(* CODESYS project Cooking chamber.project

Project tree, tasks and I/O mapping:
  Device : L-force Panel Controller p300 Logic, Lenze, order no. LPC 1000, version 3.8.0.0
    application Application
      libraries: L_PLCDataManagerAccess, 3.0.0.0 (Lenze); L_PLCLoggingAccess, 3.3.0.0 (Lenze); L_Util, 3.3.0.0 (Lenze); CAA CiA 405, 3.5.3.0 (CAA Technical Workgroup)
      task MainTask (cyclic, interval t#10ms, priority 1) calls Main
      Programs/
        program Main [ST]
        Functions/
          function Timer_convert [ST]
          function block Chamber_controller [ST]
          function block Chamber_program [ST]
          function Humidity_convert [ST]
          function block Sound_controller [ST]
          function block Alarm_controller [ST]
        Routines/
          program Controller [ST]
        System/
          program Analog_controller [ST]
      Variables/
        global variables Global
        global variables Settings
        global variables Recipes
      Symbols/
        Symbols
    CANbus : CANbus, Lenze, version 2.0.0.0
      CANopen_Manager : CANopen_Manager, Lenze, version 3.12.0.0
          settings: Sync CycleTime in Microseconds = 10000; Enable Sync generation = TRUE; Heartbeat Node ID = 63; Can Open Node ID = 63; ConfigVersion = 50659584
        EPM_S110 : EPM-S110, Lenze, order no. EPM-S110, version 1.14.0.5
            settings: General Options.Reset Node = FALSE; NODEIDSAVED = 1; SDO Timeout = 1000000; EXPERTSETTINGS = TRUE; Sync-General Parameters.Communication Cycle Period = 16#00002710 usec; Synchronous Window Length = 16#000004B0; Emergency-General Parameters.Emergency enabled = FALSE; Settings.COBID = 16#00000201; Settings.Transmission Type = 16#FF; Settings.available PDO-Parameter.Inhibit Time available = FALSE; Settings.available PDO-Parameter.Event Timer available = FALSE; Settings.Inhibit Time = 0; Settings.Event Timer = 0; Generic COBID = '$NODEID+16#0200'; Settings.COBID = 16#00000181; Settings.Transmission Type = 16#01; Settings.available PDO-Parameter.Inhibit Time available = TRUE; Settings.available PDO-Parameter.Event Timer available = TRUE; Settings.Inhibit Time = 0; Settings.Event Timer = 0; Generic COBID = '$NODEID+16#0180'; Settings.COBID = 16#00000281; Settings.Transmission Type = 16#01; Settings.available PDO-Parameter.Inhibit Time available = TRUE; Settings.available PDO-Parameter.Event Timer available = TRUE; Settings.Inhibit Time = 0; Settings.Event Timer = 0; Generic COBID = '$NODEID+16#0280'; Settings.COBID = 16#00000381; Settings.Transmission Type = 16#01; Settings.available PDO-Parameter.Inhibit Time available = TRUE; Settings.available PDO-Parameter.Event Timer available = TRUE; Settings.Inhibit Time = 0; Settings.Event Timer = 0; Generic COBID = '$NODEID+16#0380'; Setting /state digital Output : EPM_S302_DO8_DC24V_5A_02.Index = 16#6200; Setting /state digital Output : EPM_S302_DO8_DC24V_5A_02.Subindex = 16#01; Setting /state digital Output : EPM_S302_DO8_DC24V_5A_02.ObjectLength = 8; Setting /state digital Output : EPM_S302_DO8_DC24V_5A_03.Index = 16#6200; Setting /state digital Output : EPM_S302_DO8_DC24V_5A_03.Subindex = 16#02;
              Setting /state digital Output : EPM_S302_DO8_DC24V_5A_03.ObjectLength = 8; State digital input : EPM_S202_DI8_DC24V_00.Index = 16#6000; State digital input : EPM_S202_DI8_DC24V_00.Subindex = 16#01; State digital input : EPM_S202_DI8_DC24V_00.ObjectLength = 8; State digital input : EPM_S202_DI8_DC24V_01.Index = 16#6000; State digital input : EPM_S202_DI8_DC24V_01.Subindex = 16#02; State digital input : EPM_S202_DI8_DC24V_01.ObjectLength = 8; Read analog Input : EPM_S404_AI4_16Bit_Resistor_04.Index = 16#6401; Read analog Input : EPM_S404_AI4_16Bit_Resistor_04.Subindex = 16#01; Read analog Input : EPM_S404_AI4_16Bit_Resistor_04.ObjectLength = 16; Read analog Input : EPM_S404_AI4_16Bit_Resistor_04.Index = 16#6401; Read analog Input : EPM_S404_AI4_16Bit_Resistor_04.Subindex = 16#02; Read analog Input : EPM_S404_AI4_16Bit_Resistor_04.ObjectLength = 16; Read analog Input : EPM_S404_AI4_16Bit_Resistor_04.Index = 16#6401; Read analog Input : EPM_S404_AI4_16Bit_Resistor_04.Subindex = 16#03; Read analog Input : EPM_S404_AI4_16Bit_Resistor_04.ObjectLength = 16; Read analog Input : EPM_S404_AI4_16Bit_Resistor_04.Index = 16#6401; Read analog Input : EPM_S404_AI4_16Bit_Resistor_04.Subindex = 16#04; Read analog Input : EPM_S404_AI4_16Bit_Resistor_04.ObjectLength = 16; Read analog Input : EPM_S404_AI4_16Bit_Resistor_05.Index = 16#6401; Read analog Input : EPM_S404_AI4_16Bit_Resistor_05.Subindex = 16#05; Read analog Input : EPM_S404_AI4_16Bit_Resistor_05.ObjectLength = 16; Read analog Input : EPM_S404_AI4_16Bit_Resistor_05.Index = 16#6401; Read analog Input : EPM_S404_AI4_16Bit_Resistor_05.Subindex = 16#06; Read analog Input : EPM_S404_AI4_16Bit_Resistor_05.ObjectLength = 16; Read analog Input : EPM_S404_AI4_16Bit_Resistor_05.Index = 16#6401; Read analog Input : EPM_S404_AI4_16Bit_Resistor_05.Subindex = 16#07; Read analog Input : EPM_S404_AI4_16Bit_Resistor_05.ObjectLength = 16; Read analog Input : EPM_S404_AI4_16Bit_Resistor_05.Index = 16#6401; Read analog Input : EPM_S404_AI4_16Bit_Resistor_05.Subindex = 16#08; Read analog Input : EPM_S404_AI4_16Bit_Resistor_05.ObjectLength = 16; SDO List.Set COB-ID sync.Index = 16#1005; SDO List.Set COB-ID sync.Subindex = 16#00; SDO List.Set COB-ID sync.Value = 16#80000080; SDO List.Set COB-ID sync.Size = 32; SDO List.Set COB-ID sync.AbortIfError = FALSE; SDO List.Set COB-ID sync.JumpToLine = FALSE; SDO List.Set COB-ID sync.Line = 0; SDO List.Set synchronous window length.Index = 16#1007; SDO List.Set synchronous window length.Subindex = 16#00;
              SDO List.Set synchronous window length.Value = 16#000004B0; SDO List.Set synchronous window length.Size = 32; SDO List.Set synchronous window length.AbortIfError = FALSE; SDO List.Set synchronous window length.JumpToLine = FALSE; SDO List.Set synchronous window length.Line = 0; SDO List.Set Guardtime.Index = 16#100C; SDO List.Set Guardtime.Subindex = 16#00; SDO List.Set Guardtime.Value = 16#00000000; SDO List.Set Guardtime.Size = 16; SDO List.Set Guardtime.AbortIfError = FALSE; SDO List.Set Guardtime.JumpToLine = FALSE; SDO List.Set Guardtime.Line = 0; SDO List.Set Lifetime.Index = 16#100D; SDO List.Set Lifetime.Subindex = 16#00; SDO List.Set Lifetime.Value = 16#00000000; SDO List.Set Lifetime.Size = 8; SDO List.Set Lifetime.AbortIfError = FALSE; SDO List.Set Lifetime.JumpToLine = FALSE; SDO List.Set Lifetime.Line = 0; SDO List.Set Heartbeat Consumer.Index = 16#1016; SDO List.Set Heartbeat Consumer.Subindex = 16#01; SDO List.Set Heartbeat Consumer.Value = 0; SDO List.Set Heartbeat Consumer.Size = 32; SDO List.Set Heartbeat Consumer.AbortIfError = FALSE; SDO List.Set Heartbeat Consumer.JumpToLine = FALSE; SDO List.Set Heartbeat Consumer.Line = 0; SDO List.Set Heartbeat Consumer.Index = 16#1016; SDO List.Set Heartbeat Consumer.Subindex = 16#02; SDO List.Set Heartbeat Consumer.Value = 0; SDO List.Set Heartbeat Consumer.Size = 32; SDO List.Set Heartbeat Consumer.AbortIfError = FALSE; SDO List.Set Heartbeat Consumer.JumpToLine = FALSE; SDO List.Set Heartbeat Consumer.Line = 0; SDO List.Set Heartbeat Consumer.Index = 16#1016; SDO List.Set Heartbeat Consumer.Subindex = 16#03; SDO List.Set Heartbeat Consumer.Value = 0; SDO List.Set Heartbeat Consumer.Size = 32; SDO List.Set Heartbeat Consumer.AbortIfError = FALSE; SDO List.Set Heartbeat Consumer.JumpToLine = FALSE; SDO List.Set Heartbeat Consumer.Line = 0;
              SDO List.Set Heartbeat Consumer.Index = 16#1016; SDO List.Set Heartbeat Consumer.Subindex = 16#04; SDO List.Set Heartbeat Consumer.Value = 0; SDO List.Set Heartbeat Consumer.Size = 32; SDO List.Set Heartbeat Consumer.AbortIfError = FALSE; SDO List.Set Heartbeat Consumer.JumpToLine = FALSE; SDO List.Set Heartbeat Consumer.Line = 0; SDO List.Set Heartbeat Consumer.Index = 16#1016; SDO List.Set Heartbeat Consumer.Subindex = 16#05; SDO List.Set Heartbeat Consumer.Value = 0; SDO List.Set Heartbeat Consumer.Size = 32; SDO List.Set Heartbeat Consumer.AbortIfError = FALSE; SDO List.Set Heartbeat Consumer.JumpToLine = FALSE; SDO List.Set Heartbeat Consumer.Line = 0; SDO List.Set Heartbeat Producer.Index = 16#1017; SDO List.Set Heartbeat Producer.Subindex = 16#00; SDO List.Set Heartbeat Producer.Value = 16#00000000; SDO List.Set Heartbeat Producer.Size = 16; SDO List.Set Heartbeat Producer.AbortIfError = FALSE; SDO List.Set Heartbeat Producer.JumpToLine = FALSE; SDO List.Set Heartbeat Producer.Line = 0; SDO List.Disable PDO.Index = 16#1400; SDO List.Disable PDO.Subindex = 16#01; SDO List.Disable PDO.Value = 16#80000201; SDO List.Disable PDO.Size = 32; SDO List.Disable PDO.AbortIfError = FALSE; SDO List.Disable PDO.JumpToLine = FALSE; SDO List.Disable PDO.Line = 0; SDO List.Set transmission type.Index = 16#1400; SDO List.Set transmission type.Subindex = 16#02; SDO List.Set transmission type.Value = 16#FF; SDO List.Set transmission type.Size = 8; SDO List.Set transmission type.AbortIfError = FALSE; SDO List.Set transmission type.JumpToLine = FALSE; SDO List.Set transmission type.Line = 0; SDO List.Clear pdo mapping.Index = 16#1600; SDO List.Clear pdo mapping.Subindex = 16#00; SDO List.Clear pdo mapping.Value = 16#0; SDO List.Clear pdo mapping.Size = 8; SDO List.Clear pdo mapping.AbortIfError = FALSE;
              SDO List.Clear pdo mapping.JumpToLine = FALSE; SDO List.Clear pdo mapping.Line = 0; SDO List.Set Mapping.Index = 16#1600; SDO List.Set Mapping.Subindex = 16#01; SDO List.Set Mapping.Value = 16#62000108; SDO List.Set Mapping.Size = 32; SDO List.Set Mapping.AbortIfError = FALSE; SDO List.Set Mapping.JumpToLine = FALSE; SDO List.Set Mapping.Line = 0; SDO List.Set Mapping.Index = 16#1600; SDO List.Set Mapping.Subindex = 16#02; SDO List.Set Mapping.Value = 16#62000208; SDO List.Set Mapping.Size = 32; SDO List.Set Mapping.AbortIfError = FALSE; SDO List.Set Mapping.JumpToLine = FALSE; SDO List.Set Mapping.Line = 0; SDO List.Set number of mappings.Index = 16#1600; SDO List.Set number of mappings.Subindex = 16#00; SDO List.Set number of mappings.Value = 16#02; SDO List.Set number of mappings.Size = 8; SDO List.Set number of mappings.AbortIfError = FALSE; SDO List.Set number of mappings.JumpToLine = FALSE; SDO List.Set number of mappings.Line = 0; SDO List.Set and enable COB-ID.Index = 16#1400; SDO List.Set and enable COB-ID.Subindex = 16#01; SDO List.Set and enable COB-ID.Value = 16#00000201; SDO List.Set and enable COB-ID.Size = 32; SDO List.Set and enable COB-ID.AbortIfError = FALSE; SDO List.Set and enable COB-ID.JumpToLine = FALSE; SDO List.Set and enable COB-ID.Line = 0; SDO List.Disable PDO.Index = 16#1800; SDO List.Disable PDO.Subindex = 16#01; SDO List.Disable PDO.Value = 16#80000181; SDO List.Disable PDO.Size = 32; SDO List.Disable PDO.AbortIfError = FALSE; SDO List.Disable PDO.JumpToLine = FALSE; SDO List.Disable PDO.Line = 0; SDO List.Set transmission type.Index = 16#1800; SDO List.Set transmission type.Subindex = 16#02; SDO List.Set transmission type.Value = 16#01;
              SDO List.Set transmission type.Size = 8; SDO List.Set transmission type.AbortIfError = FALSE; SDO List.Set transmission type.JumpToLine = FALSE; SDO List.Set transmission type.Line = 0; SDO List.Set inhibit time.Index = 16#1800; SDO List.Set inhibit time.Subindex = 16#03; SDO List.Set inhibit time.Value = 16#0000; SDO List.Set inhibit time.Size = 16; SDO List.Set inhibit time.AbortIfError = FALSE; SDO List.Set inhibit time.JumpToLine = FALSE; SDO List.Set inhibit time.Line = 0; SDO List.Set event time.Index = 16#1800; SDO List.Set event time.Subindex = 16#05; SDO List.Set event time.Value = 16#0000; SDO List.Set event time.Size = 16; SDO List.Set event time.AbortIfError = FALSE; SDO List.Set event time.JumpToLine = FALSE; SDO List.Set event time.Line = 0; SDO List.Clear pdo mapping.Index = 16#1A00; SDO List.Clear pdo mapping.Subindex = 16#00; SDO List.Clear pdo mapping.Value = 16#0; SDO List.Clear pdo mapping.Size = 8; SDO List.Clear pdo mapping.AbortIfError = FALSE; SDO List.Clear pdo mapping.JumpToLine = FALSE; SDO List.Clear pdo mapping.Line = 0; SDO List.Set Mapping.Index = 16#1A00; SDO List.Set Mapping.Subindex = 16#01; SDO List.Set Mapping.Value = 16#60000108; SDO List.Set Mapping.Size = 32; SDO List.Set Mapping.AbortIfError = FALSE; SDO List.Set Mapping.JumpToLine = FALSE; SDO List.Set Mapping.Line = 0; SDO List.Set Mapping.Index = 16#1A00; SDO List.Set Mapping.Subindex = 16#02; SDO List.Set Mapping.Value = 16#60000208; SDO List.Set Mapping.Size = 32; SDO List.Set Mapping.AbortIfError = FALSE; SDO List.Set Mapping.JumpToLine = FALSE; SDO List.Set Mapping.Line = 0; SDO List.Set number of mappings.Index = 16#1A00;
              SDO List.Set number of mappings.Subindex = 16#00; SDO List.Set number of mappings.Value = 16#02; SDO List.Set number of mappings.Size = 8; SDO List.Set number of mappings.AbortIfError = FALSE; SDO List.Set number of mappings.JumpToLine = FALSE; SDO List.Set number of mappings.Line = 0; SDO List.Set and enable COB-ID.Index = 16#1800; SDO List.Set and enable COB-ID.Subindex = 16#01; SDO List.Set and enable COB-ID.Value = 16#00000181; SDO List.Set and enable COB-ID.Size = 32; SDO List.Set and enable COB-ID.AbortIfError = FALSE; SDO List.Set and enable COB-ID.JumpToLine = FALSE; SDO List.Set and enable COB-ID.Line = 0; SDO List.Disable PDO.Index = 16#1801; SDO List.Disable PDO.Subindex = 16#01; SDO List.Disable PDO.Value = 16#80000281; SDO List.Disable PDO.Size = 32; SDO List.Disable PDO.AbortIfError = FALSE; SDO List.Disable PDO.JumpToLine = FALSE; SDO List.Disable PDO.Line = 0; SDO List.Set transmission type.Index = 16#1801; SDO List.Set transmission type.Subindex = 16#02; SDO List.Set transmission type.Value = 16#01; SDO List.Set transmission type.Size = 8; SDO List.Set transmission type.AbortIfError = FALSE; SDO List.Set transmission type.JumpToLine = FALSE; SDO List.Set transmission type.Line = 0; SDO List.Set inhibit time.Index = 16#1801; SDO List.Set inhibit time.Subindex = 16#03; SDO List.Set inhibit time.Value = 16#0000; SDO List.Set inhibit time.Size = 16; SDO List.Set inhibit time.AbortIfError = FALSE; SDO List.Set inhibit time.JumpToLine = FALSE; SDO List.Set inhibit time.Line = 0; SDO List.Set event time.Index = 16#1801; SDO List.Set event time.Subindex = 16#05; SDO List.Set event time.Value = 16#0000; SDO List.Set event time.Size = 16; SDO List.Set event time.AbortIfError = FALSE; SDO List.Set event time.JumpToLine = FALSE;
              SDO List.Set event time.Line = 0; SDO List.Clear pdo mapping.Index = 16#1A01; SDO List.Clear pdo mapping.Subindex = 16#00; SDO List.Clear pdo mapping.Value = 16#0; SDO List.Clear pdo mapping.Size = 8; SDO List.Clear pdo mapping.AbortIfError = FALSE; SDO List.Clear pdo mapping.JumpToLine = FALSE; SDO List.Clear pdo mapping.Line = 0; SDO List.Set Mapping.Index = 16#1A01; SDO List.Set Mapping.Subindex = 16#01; SDO List.Set Mapping.Value = 16#64010110; SDO List.Set Mapping.Size = 32; SDO List.Set Mapping.AbortIfError = FALSE; SDO List.Set Mapping.JumpToLine = FALSE; SDO List.Set Mapping.Line = 0; SDO List.Set Mapping.Index = 16#1A01; SDO List.Set Mapping.Subindex = 16#02; SDO List.Set Mapping.Value = 16#64010210; SDO List.Set Mapping.Size = 32; SDO List.Set Mapping.AbortIfError = FALSE; SDO List.Set Mapping.JumpToLine = FALSE; SDO List.Set Mapping.Line = 0; SDO List.Set Mapping.Index = 16#1A01; SDO List.Set Mapping.Subindex = 16#03; SDO List.Set Mapping.Value = 16#64010310; SDO List.Set Mapping.Size = 32; SDO List.Set Mapping.AbortIfError = FALSE; SDO List.Set Mapping.JumpToLine = FALSE; SDO List.Set Mapping.Line = 0; SDO List.Set Mapping.Index = 16#1A01; SDO List.Set Mapping.Subindex = 16#04; SDO List.Set Mapping.Value = 16#64010410; SDO List.Set Mapping.Size = 32; SDO List.Set Mapping.AbortIfError = FALSE; SDO List.Set Mapping.JumpToLine = FALSE; SDO List.Set Mapping.Line = 0; SDO List.Set number of mappings.Index = 16#1A01; SDO List.Set number of mappings.Subindex = 16#00; SDO List.Set number of mappings.Value = 16#04; SDO List.Set number of mappings.Size = 8;
              SDO List.Set number of mappings.AbortIfError = FALSE; SDO List.Set number of mappings.JumpToLine = FALSE; SDO List.Set number of mappings.Line = 0; SDO List.Set and enable COB-ID.Index = 16#1801; SDO List.Set and enable COB-ID.Subindex = 16#01; SDO List.Set and enable COB-ID.Value = 16#00000281; SDO List.Set and enable COB-ID.Size = 32; SDO List.Set and enable COB-ID.AbortIfError = FALSE; SDO List.Set and enable COB-ID.JumpToLine = FALSE; SDO List.Set and enable COB-ID.Line = 0; SDO List.Disable PDO.Index = 16#1802; SDO List.Disable PDO.Subindex = 16#01; SDO List.Disable PDO.Value = 16#80000381; SDO List.Disable PDO.Size = 32; SDO List.Disable PDO.AbortIfError = FALSE; SDO List.Disable PDO.JumpToLine = FALSE; SDO List.Disable PDO.Line = 0; SDO List.Set transmission type.Index = 16#1802; SDO List.Set transmission type.Subindex = 16#02; SDO List.Set transmission type.Value = 16#01; SDO List.Set transmission type.Size = 8; SDO List.Set transmission type.AbortIfError = FALSE; SDO List.Set transmission type.JumpToLine = FALSE; SDO List.Set transmission type.Line = 0; SDO List.Set inhibit time.Index = 16#1802; SDO List.Set inhibit time.Subindex = 16#03; SDO List.Set inhibit time.Value = 16#0000; SDO List.Set inhibit time.Size = 16; SDO List.Set inhibit time.AbortIfError = FALSE; SDO List.Set inhibit time.JumpToLine = FALSE; SDO List.Set inhibit time.Line = 0; SDO List.Set event time.Index = 16#1802; SDO List.Set event time.Subindex = 16#05; SDO List.Set event time.Value = 16#0000; SDO List.Set event time.Size = 16; SDO List.Set event time.AbortIfError = FALSE; SDO List.Set event time.JumpToLine = FALSE; SDO List.Set event time.Line = 0; SDO List.Clear pdo mapping.Index = 16#1A02; SDO List.Clear pdo mapping.Subindex = 16#00;
              SDO List.Clear pdo mapping.Value = 16#0; SDO List.Clear pdo mapping.Size = 8; SDO List.Clear pdo mapping.AbortIfError = FALSE; SDO List.Clear pdo mapping.JumpToLine = FALSE; SDO List.Clear pdo mapping.Line = 0; SDO List.Set Mapping.Index = 16#1A02; SDO List.Set Mapping.Subindex = 16#01; SDO List.Set Mapping.Value = 16#64010510; SDO List.Set Mapping.Size = 32; SDO List.Set Mapping.AbortIfError = FALSE; SDO List.Set Mapping.JumpToLine = FALSE; SDO List.Set Mapping.Line = 0; SDO List.Set Mapping.Index = 16#1A02; SDO List.Set Mapping.Subindex = 16#02; SDO List.Set Mapping.Value = 16#64010610; SDO List.Set Mapping.Size = 32; SDO List.Set Mapping.AbortIfError = FALSE; SDO List.Set Mapping.JumpToLine = FALSE; SDO List.Set Mapping.Line = 0; SDO List.Set Mapping.Index = 16#1A02; SDO List.Set Mapping.Subindex = 16#03; SDO List.Set Mapping.Value = 16#64010710; SDO List.Set Mapping.Size = 32; SDO List.Set Mapping.AbortIfError = FALSE; SDO List.Set Mapping.JumpToLine = FALSE; SDO List.Set Mapping.Line = 0; SDO List.Set Mapping.Index = 16#1A02; SDO List.Set Mapping.Subindex = 16#04; SDO List.Set Mapping.Value = 16#64010810; SDO List.Set Mapping.Size = 32; SDO List.Set Mapping.AbortIfError = FALSE; SDO List.Set Mapping.JumpToLine = FALSE; SDO List.Set Mapping.Line = 0; SDO List.Set number of mappings.Index = 16#1A02; SDO List.Set number of mappings.Subindex = 16#00; SDO List.Set number of mappings.Value = 16#04; SDO List.Set number of mappings.Size = 8; SDO List.Set number of mappings.AbortIfError = FALSE; SDO List.Set number of mappings.JumpToLine = FALSE; SDO List.Set number of mappings.Line = 0;
              SDO List.Set and enable COB-ID.Index = 16#1802; SDO List.Set and enable COB-ID.Subindex = 16#01; SDO List.Set and enable COB-ID.Value = 16#00000381; SDO List.Set and enable COB-ID.Size = 32; SDO List.Set and enable COB-ID.AbortIfError = FALSE; SDO List.Set and enable COB-ID.JumpToLine = FALSE; SDO List.Set and enable COB-ID.Line = 0; ConfigVersion = 50659584
          EPM_S202_DI8_DC24V_00 : EPM-S202 DI8, DC24V, Lenze, order no. EPM-S202, version 1.14.0.5
              settings: Number of Params = 1; State digital input : EPM_S202_DI8_DC24V_00.Index = 16#6000; State digital input : EPM_S202_DI8_DC24V_00.Subindex = 16#01; State digital input : EPM_S202_DI8_DC24V_00.Startbit = 0; State digital input : EPM_S202_DI8_DC24V_00.Endbit = 7
              input  Application.Emergency_chamber[00] : BOOL  // State digital input : EPM_S202_DI8_DC24V_00.Bit0
              input  Application.Motor_protection[00] : BOOL  // State digital input : EPM_S202_DI8_DC24V_00.Bit1
              input  Application.Burner_protection[00] : BOOL  // State digital input : EPM_S202_DI8_DC24V_00.Bit2
              unmapped channels: State digital input : EPM_S202_DI8_DC24V_00
          EPM_S202_DI8_DC24V_01 : EPM-S202 DI8, DC24V, Lenze, order no. EPM-S202, version 1.14.0.5
              settings: Number of Params = 1; State digital input : EPM_S202_DI8_DC24V_01.Index = 16#6000; State digital input : EPM_S202_DI8_DC24V_01.Subindex = 16#02; State digital input : EPM_S202_DI8_DC24V_01.Startbit = 0; State digital input : EPM_S202_DI8_DC24V_01.Endbit = 7
              input  Application.Emergency_chamber[01] : BOOL  // State digital input : EPM_S202_DI8_DC24V_01.Bit0
              input  Application.Motor_protection[01] : BOOL  // State digital input : EPM_S202_DI8_DC24V_01.Bit1
              input  Application.Burner_protection[01] : BOOL  // State digital input : EPM_S202_DI8_DC24V_01.Bit2
              unmapped channels: State digital input : EPM_S202_DI8_DC24V_01
          EPM_S302_DO8_DC24V_5A_02 : EPM-S302 DO8, DC24V, 0,5A, Lenze, order no. EPM-S302, version 1.14.0.5
              settings: Number of Params = 1; Setting /state digital Output : EPM_S302_DO8_DC24V_5A_02.Index = 16#6200; Setting /state digital Output : EPM_S302_DO8_DC24V_5A_02.Subindex = 16#01; Setting /state digital Output : EPM_S302_DO8_DC24V_5A_02.Startbit = 0; Setting /state digital Output : EPM_S302_DO8_DC24V_5A_02.Endbit = 7
              output Application.Burner_activation[00] : BOOL  // Setting /state digital Output : EPM_S302_DO8_DC24V_5A_02.Bit0
              output Application.Burner_reset[00] : BOOL  // Setting /state digital Output : EPM_S302_DO8_DC24V_5A_02.Bit1
              output Application.Chimney_activation[00] : BOOL  // Setting /state digital Output : EPM_S302_DO8_DC24V_5A_02.Bit2
              output Application.Smokehouse_activation[00] : BOOL  // Setting /state digital Output : EPM_S302_DO8_DC24V_5A_02.Bit3
              output Application.Beeb_activation : BOOL  // Setting /state digital Output : EPM_S302_DO8_DC24V_5A_02.Bit4
              output Application.Motor_activation[00, 00] : BOOL  // Setting /state digital Output : EPM_S302_DO8_DC24V_5A_02.Bit5
              output Application.Motor_activation[00, 01] : BOOL  // Setting /state digital Output : EPM_S302_DO8_DC24V_5A_02.Bit6
              output Application.Motor_activation[00, 02] : BOOL  // Setting /state digital Output : EPM_S302_DO8_DC24V_5A_02.Bit7
              unmapped channels: Setting /state digital Output : EPM_S302_DO8_DC24V_5A_02
          EPM_S302_DO8_DC24V_5A_03 : EPM-S302 DO8, DC24V, 0,5A, Lenze, order no. EPM-S302, version 1.14.0.5
              settings: Number of Params = 1; Setting /state digital Output : EPM_S302_DO8_DC24V_5A_03.Index = 16#6200; Setting /state digital Output : EPM_S302_DO8_DC24V_5A_03.Subindex = 16#02; Setting /state digital Output : EPM_S302_DO8_DC24V_5A_03.Startbit = 0; Setting /state digital Output : EPM_S302_DO8_DC24V_5A_03.Endbit = 7
              output Application.Burner_activation[01] : BOOL  // Setting /state digital Output : EPM_S302_DO8_DC24V_5A_03.Bit0
              output Application.Burner_reset[01] : BOOL  // Setting /state digital Output : EPM_S302_DO8_DC24V_5A_03.Bit1
              output Application.Chimney_activation[01] : BOOL  // Setting /state digital Output : EPM_S302_DO8_DC24V_5A_03.Bit2
              output Application.Smokehouse_activation[01] : BOOL  // Setting /state digital Output : EPM_S302_DO8_DC24V_5A_03.Bit3
              output Application.Motor_activation[01, 00] : BOOL  // Setting /state digital Output : EPM_S302_DO8_DC24V_5A_03.Bit5
              output Application.Motor_activation[01, 01] : BOOL  // Setting /state digital Output : EPM_S302_DO8_DC24V_5A_03.Bit6
              output Application.Motor_activation[01, 02] : BOOL  // Setting /state digital Output : EPM_S302_DO8_DC24V_5A_03.Bit7
              unmapped channels: Setting /state digital Output : EPM_S302_DO8_DC24V_5A_03
          EPM_S404_AI4_16Bit_Resistor_04 : EPM-S404 AI4 16Bit, Resistor, Lenze, order no. EPM-S404, version 1.14.0.5
              settings: Number of Params = 4; Read analog Input : EPM_S404_AI4_16Bit_Resistor_04.Index = 16#6401; Read analog Input : EPM_S404_AI4_16Bit_Resistor_04.Subindex = 16#01; Read analog Input : EPM_S404_AI4_16Bit_Resistor_04.Startbit = 0; Read analog Input : EPM_S404_AI4_16Bit_Resistor_04.Endbit = 15; Read analog Input : EPM_S404_AI4_16Bit_Resistor_04.Index = 16#6401; Read analog Input : EPM_S404_AI4_16Bit_Resistor_04.Subindex = 16#02; Read analog Input : EPM_S404_AI4_16Bit_Resistor_04.Startbit = 0; Read analog Input : EPM_S404_AI4_16Bit_Resistor_04.Endbit = 15; Read analog Input : EPM_S404_AI4_16Bit_Resistor_04.Index = 16#6401; Read analog Input : EPM_S404_AI4_16Bit_Resistor_04.Subindex = 16#03; Read analog Input : EPM_S404_AI4_16Bit_Resistor_04.Startbit = 0; Read analog Input : EPM_S404_AI4_16Bit_Resistor_04.Endbit = 15; Read analog Input : EPM_S404_AI4_16Bit_Resistor_04.Index = 16#6401; Read analog Input : EPM_S404_AI4_16Bit_Resistor_04.Subindex = 16#04; Read analog Input : EPM_S404_AI4_16Bit_Resistor_04.Startbit = 0; Read analog Input : EPM_S404_AI4_16Bit_Resistor_04.Endbit = 15
              input  Application.Core_temperature_sensor[00] : WORD  // Read analog Input : EPM_S404_AI4_16Bit_Resistor_04
              input  Application.Chamber_temperature_dry_sensor[00] : WORD  // Read analog Input : EPM_S404_AI4_16Bit_Resistor_04
              input  Application.Core_temperature_sensor[01] : WORD  // Read analog Input : EPM_S404_AI4_16Bit_Resistor_04
              input  Application.Chamber_temperature_dry_sensor[01] : WORD  // Read analog Input : EPM_S404_AI4_16Bit_Resistor_04
          EPM_S404_AI4_16Bit_Resistor_05 : EPM-S404 AI4 16Bit, Resistor, Lenze, order no. EPM-S404, version 1.14.0.5
              settings: Number of Params = 4; Read analog Input : EPM_S404_AI4_16Bit_Resistor_05.Index = 16#6401; Read analog Input : EPM_S404_AI4_16Bit_Resistor_05.Subindex = 16#05; Read analog Input : EPM_S404_AI4_16Bit_Resistor_05.Startbit = 0; Read analog Input : EPM_S404_AI4_16Bit_Resistor_05.Endbit = 15; Read analog Input : EPM_S404_AI4_16Bit_Resistor_05.Index = 16#6401; Read analog Input : EPM_S404_AI4_16Bit_Resistor_05.Subindex = 16#06; Read analog Input : EPM_S404_AI4_16Bit_Resistor_05.Startbit = 0; Read analog Input : EPM_S404_AI4_16Bit_Resistor_05.Endbit = 15; Read analog Input : EPM_S404_AI4_16Bit_Resistor_05.Index = 16#6401; Read analog Input : EPM_S404_AI4_16Bit_Resistor_05.Subindex = 16#07; Read analog Input : EPM_S404_AI4_16Bit_Resistor_05.Startbit = 0; Read analog Input : EPM_S404_AI4_16Bit_Resistor_05.Endbit = 15; Read analog Input : EPM_S404_AI4_16Bit_Resistor_05.Index = 16#6401; Read analog Input : EPM_S404_AI4_16Bit_Resistor_05.Subindex = 16#08; Read analog Input : EPM_S404_AI4_16Bit_Resistor_05.Startbit = 0; Read analog Input : EPM_S404_AI4_16Bit_Resistor_05.Endbit = 15
              unmapped channels: Read analog Input : EPM_S404_AI4_16Bit_Resistor_05, Read analog Input : EPM_S404_AI4_16Bit_Resistor_05, Read analog Input : EPM_S404_AI4_16Bit_Resistor_05, Read analog Input : EPM_S404_AI4_16Bit_Resistor_05
*)

// Device/Application/Variables/Global
VAR_GLOBAL
			
	//Chamber controller
	
		// Emergency control chamber
			Emergency_chamber: ARRAY [00..02] OF BOOL := [3(0)];

		// Core product temperature sensor
			Core_temperature_sensor: ARRAY [00..02] OF WORD := [3(0)];
		
		// Core product temperature
			Core_temperature: ARRAY [00..02] OF REAL := [3(0)];
		
		// Temperature sensor dry of the chamber
			Chamber_temperature_dry_sensor: ARRAY [00..02] OF WORD := [3(0)];
		
		// Temperature sensor wet of the chamber
			Chamber_temperature_wet_sensor: ARRAY [00..02] OF WORD := [3(0)];
			
		// Temperature chamber
			Chamber_temperature: ARRAY [00..02] OF REAL := [3(0)];
		
		// Humidity chamber
			Chamber_humidity: ARRAY [00..02] OF INT := [3(0)];
			
		// Burner protection circuit
			Burner_protection: ARRAY [00..02] OF BOOL := [3(0)];
	
		// Activation burner
			Burner_activation: ARRAY [00..02] OF BOOL := [3(0)];
		
		// Reset burner
			Burner_reset: ARRAY [00..02] OF BOOL := [3(0)];
		
		// Motor protection circuit
			Motor_protection: ARRAY [00..02] OF BOOL := [3(0)];
			
		// Activation motor
			Motor_activation: ARRAY [00..02, 00..10] OF BOOL := [10(0), 10(0), 10(0)];
		
		// Activation of the steam valve
			Steam_valve_activation: ARRAY [00..02] OF BOOL := [3(0)];
			
		// Activation of the humidification valve
			Humidification_valve_activation: ARRAY [00..02] OF BOOL := [3(0)];
		
		// Activation chimney
			Chimney_activation: ARRAY [00..02] OF BOOL := [3(0)];
		
		// Higher chimney closed
			Higher_chimney_closed: ARRAY [00..02] OF BOOL := [3(0)];
		
		// Higher chimney open	
			Higher_chimney_open: ARRAY [00..02] OF BOOL := [3(0)];
		
		// Lower chimney closed	
			Lower_chimney_closed: ARRAY [00..02] OF BOOL := [3(0)];
		
		// Lower chimney open
			Lower_chimney_open: ARRAY [00..02] OF BOOL := [3(0)];
		
		// Smokehouse protection circuit
			Smokehouse_protection: ARRAY [00..02] OF BOOL := [3(0)];
			
		// Activation smokehouse
			Smokehouse_activation: ARRAY [00..02] OF BOOL := [3(0)];
		
		// Activation sound
			Sound_activation: ARRAY [00..02] OF BOOL := [3(0)];
		
		// Activation beeb
			Beeb_activation: BOOL := 0;
	
		// Chambers alarms status
			Alarms_chambers_status: ARRAY [00..02] OF INT := [3(0)];
			
		// Alarms acknowledge
			Alamrs_acknowledge: BOOL := FALSE;
			
		// Alarms activation
			Alarms_activation: BOOL := FALSE;
			
	// Program chamber
	
		// Programm recipe chamber
			Program_recipe_chamber: INT := 0;	
			
		// Programm chamber
			Program_chamber: ARRAY [00..02] OF BOOL := [3(0)];;
			
		// Programm chamber status
			Program_chamber_status: ARRAY [00..02] OF INT := [3(0)];
			
		// Programm cycles
			Program_cycles: ARRAY [00..02] OF INT := [3(0)];
			
		// Programm steps
			Program_steps: ARRAY [00..02] OF INT := [3(0)];
		
		// Program estimated
			Program_estimated: ARRAY [00..02] OF INT := [3(0)];
			
		// Program elapsed
			Program_elapsed: ARRAY [00..02] OF INT := [3(0)];
	
		// Program estimated time
			Program_estimated_time: ARRAY [00..02] OF DATE_AND_TIME := [3(DT#1970-01-01-00:00:00)];
			
		// Program prcocess init
			Program_process_init: ARRAY [00..02] OF DATE_AND_TIME := [3(DT#1970-01-01-00:00:00)];
		
END_VAR

// Device/Application/Variables/Settings
VAR_GLOBAL PERSISTENT RETAIN
	
	// Limits
	
		// Lower limit of temperature
			Lower_limit_temperature: REAL := 25.0;
			
		// Upper limit of temperature
			Upper_limit_temperature: REAL := 250.0;
			
		// Lower limmit of timer cycle
			Lower_limit_timer_cycle: INT := 1;
			
		// Upper limit of timer cycle
			Upper_limit_timer_cycle: INT := 1000;
			
		// Lower limit of humidity
			lower_limit_humidity: INT := 1;
			
		// Upper limit of humidity
			Upper_limit_humidity: INT := 99;
			
	// Calibration
	
		// Core product temperature sensor offset
			Core_temperature_offset: ARRAY [00..02] OF REAL := [3(0.0)];
		
		// Temperature chamber offset
			Chamber_temperature_offset: ARRAY [00..02] OF REAL := [3(0.0)];
		
		// Humidity chamber offset
			Chamber_humidity_offset: ARRAY [00..02] OF INT := [3(0)];
			
	// System
	
		// Temperature maximum
			Temperature_maximum: REAL := 300.0;
			
		// Temperature control system
			Temperature_control_system: BOOL := FALSE;
			
		// Enabled chambers
			Enabled_chambers: INT := 2;
			
		// Enabled chamber cars
			Enabled_chamber_cars: INT := 4;
			
	// Timers
	
		// Timer activation motors
			Timer_activation_motors: INT := 10;
			
		// Timer activation humidification valve
			Timer_activation_humidification_valve: INT := 5;
			
		// Timer response humidification valve
			timer_response_humidification_valve: INT:= 5;
			
	// Hysteresis
	
		// Temperature upper hysteresis
			Temperature_upper_hysteresis: REAL := 2.0;
			
		// Temperature lower hysteresis
			Temperature_lower_hysteresis: REAL := 2.0;
			
		// Humidity upper hysteresis
			Humidity_upper_hysteresis: INT := 2;
			
		// Humidity lower hysteresis
			Humidity_lower_hysteresis: INT := 2;
			
END_VAR

// Device/Application/Variables/Recipes
VAR_GLOBAL
	
	// Recipes transfer
	
		// Recipe transfer name
			Transfer_name: STRING := '';
			
		// Recipe transfer description
			Transfer_description: STRING := '';
		
		// Recipe transfer cycles
			Transfer_cycles: INT := 1;
		
		// Recipe transfer core temperature
			Transfer_core_temperature: REAL := Lower_limit_temperature;
		
		// Recipe transfer steps
			Transfer_steps: INT := 1;
	
		// Recipe transfer timer step
			Transfer_timer_step: ARRAY[00..09] OF INT := [10(Lower_limit_timer_cycle)];
				
		// Recipe transfer chamber temperature
			Transfer_chamber_temperature: ARRAY[00..09] OF REAL := [10(Lower_limit_temperature)];
			
		// Recipe transfer chamber humidity
			Transfer_chamber_humidity: ARRAY[00..09] OF INT := [10(lower_limit_humidity)];
			
		// Recipe transfer chamber chimney smokehouse
			Transfer_chamber_chimney: ARRAY[00..09] OF BOOL := [10(0)];
			
		// Recipe transfer chamber smokehouse
			Transfer_chamber_smokehouse: ARRAY[00..09] OF BOOL := [10(0)];
		
	// Recipes chamber	
	
		// Recipe name
			Recipe_name: ARRAY [00..02] OF STRING := [3('')];
			
		// Recipe description
			Recipe_description: ARRAY [00..02] OF STRING := [3('')];
			
		// Recipe cycles
			Recipe_cycles: ARRAY [00..02] OF INT := [3(0)];
		
		// Recipe core temperature
			Recipe_core_temperature: ARRAY [00..02] OF REAL := [3(0)];
		
		// Recipe steps
			Recipe_steps: ARRAY [00..02] OF INT := [3(0)];
	
		// Recipe timer step
			Recipe_timer_step: ARRAY[00..02, 00..09] OF INT := [10(0), 10(0), 10(0)];
				
		// Recipe chamber temperature
			Recipe_chamber_temperature: ARRAY[00..02, 00..09] OF REAL := [10(0), 10(0), 10(0)];
			
		// Recipe chamber humidity
			Recipe_chamber_humidity: ARRAY[00..02, 00..09] OF INT := [10(0), 10(0), 10(0)];
			
		// Recipe chamber chimney smokehouse
			Recipe_chamber_chimney: ARRAY[00..02, 00..09] OF BOOL := [10(0), 10(0), 10(0)];
			
		// Recipe chamber smokehouse
			Recipe_chamber_smokehouse: ARRAY[00..02, 00..09] OF BOOL := [10(0), 10(0), 10(0)];
		
END_VAR

// Device/Application/Programs/Main
PROGRAM Main
VAR
END_VAR

	
Analog_controller();
Controller();

END_PROGRAM

// Device/Application/Programs/System/Analog_controller
PROGRAM Analog_controller
VAR
END_VAR


// Calibration of the sensors

	// Core products temperature
		Core_temperature[00] := WORD_TO_REAL(Core_temperature_sensor[00]) / 10.0 + Core_temperature_offset[00];
		Core_temperature[01] := WORD_TO_REAL(Core_temperature_sensor[01]) / 10.0 + Core_temperature_offset[01];
		Core_temperature[02] := WORD_TO_REAL(Core_temperature_sensor[02]) / 10.0 + Core_temperature_offset[02];

	// Temperature chambers
		Chamber_temperature[00] := WORD_TO_REAL(Chamber_temperature_dry_sensor[00]) / 10.0 + Chamber_temperature_offset[00];
		Chamber_temperature[01] := WORD_TO_REAL(Chamber_temperature_dry_sensor[01]) / 10.0 + Chamber_temperature_offset[01];
		Chamber_temperature[02] := WORD_TO_REAL(Chamber_temperature_dry_sensor[02]) / 10.0 + Chamber_temperature_offset[02];

	// Humidity chambers
		Chamber_humidity[00] := REAL_TO_INT(Humidity_convert(WORD_TO_REAL(Chamber_temperature_wet_sensor[00]) / 10.0, WORD_TO_REAL(Chamber_temperature_dry_sensor[00]) / 10.0));
		Chamber_humidity[01] := REAL_TO_INT(Humidity_convert(WORD_TO_REAL(Chamber_temperature_wet_sensor[01]) / 10.0, WORD_TO_REAL(Chamber_temperature_dry_sensor[01]) / 10.0));
		Chamber_humidity[02] := REAL_TO_INT(Humidity_convert(WORD_TO_REAL(Chamber_temperature_wet_sensor[02]) / 10.0, WORD_TO_REAL(Chamber_temperature_dry_sensor[02]) / 10.0));

END_PROGRAM

// Device/Application/Programs/Functions/Humidity_convert
FUNCTION Humidity_convert: REAL
VAR_INPUT
	wet_bulb: REAL; //Wet bulb
	dry_bulb: REAL;	//Dry bulb
END_VAR
VAR
	a: REAL := 10;
	b: REAL := 10;
	c: REAL;
END_VAR


	a:= EXP(9.1466 - (2316 / (273 + wet_bulb))) - (0.5 * (dry_bulb - wet_bulb));
	b:= EXP(9.1466 - (2316 / (273 + dry_bulb)));
	c:= (a / b) * 100;
	
	IF c < 1 THEN
		c:= 1;
	END_IF
	
	IF c > 99 THEN
		c:= 99;
	END_IF

	Humidity_convert:= c;

END_FUNCTION

// Device/Application/Programs/Routines/Controller
PROGRAM Controller
VAR
	Transfer_recipe: Chamber_program();
	
	Chamber_00: Chamber_controller();
	Chamber_01: Chamber_controller();
	Chamber_02: Chamber_controller();
	
	Alarm_00: Alarm_controller();
	Alarm_01: Alarm_controller();
	Alarm_02: Alarm_controller();
	
	Sound: Sound_controller();
END_VAR

	
	Transfer_recipe(EN:= TRUE);
	
	Chamber_00(EN:= Enabled_chambers > 0, SL:= 00);
	Chamber_01(EN:= Enabled_chambers > 1, SL:= 01);
	Chamber_02(EN:= Enabled_chambers > 2, SL:= 02);
	
	Alarm_00(EN:= Enabled_chambers > 0, SL:= 00);
	Alarm_01(EN:= Enabled_chambers > 1, SL:= 01);
	Alarm_02(EN:= Enabled_chambers > 2, SL:= 02);
	
	Sound(EN:= TRUE);

END_PROGRAM

// Device/Application/Programs/Functions/Chamber_program
FUNCTION_BLOCK Chamber_program

VAR_INPUT
	EN: BOOL;	//Enable function
END_VAR

VAR_OUTPUT
END_VAR

VAR
	SL: INT;
	iCounter: INT;
	jCounter: INT;
	iEstimated: INT;
END_VAR


IF EN = TRUE THEN
	
	SL:= Program_recipe_chamber;
	
	IF SL > 0 THEN
		Recipe_name[SL -1]:= Transfer_name;
		Recipe_description[SL -1]:= Transfer_description;
		Recipe_cycles[SL - 1]:= Transfer_cycles;
		Recipe_core_temperature[SL - 1]:= Transfer_core_temperature;
		Recipe_steps[SL - 1]:= Transfer_steps;
		
		FOR iCounter:= 0 TO 9 BY 1 DO
			Recipe_timer_step[SL - 1, iCounter]:= Transfer_timer_step[iCounter];
			Recipe_chamber_temperature[SL - 1, iCounter]:= Transfer_chamber_temperature[iCounter];
			Recipe_chamber_humidity[SL - 1, iCounter]:= Transfer_chamber_humidity[iCounter];
			Recipe_chamber_chimney[SL - 1, iCounter]:= Transfer_chamber_chimney[iCounter];
			Recipe_chamber_smokehouse[SL - 1, iCounter]:= Transfer_chamber_smokehouse[iCounter];
		END_FOR
	
		iEstimated:= 0;
		
		FOR iCounter:= 0 TO Recipe_cycles[SL - 1] - 1 BY 1 DO
			
			FOR jCounter:= 0 TO Recipe_steps[SL - 1] - 1 BY 1 DO
				iEstimated:= iEstimated + Recipe_timer_step[SL - 1, jCounter];
			END_FOR
	
		END_FOR
		
		Program_estimated[SL - 1]:= iEstimated;	
		Program_recipe_chamber:= 0;	
	END_IF
	
END_IF

END_FUNCTION_BLOCK

// Device/Application/Programs/Functions/Chamber_controller
FUNCTION_BLOCK Chamber_controller

VAR_INPUT
	EN: BOOL;	//Enable function
	SL: INT;	//Index of the chamber
END_VAR

VAR_OUTPUT
END_VAR

VAR
	iEsti: LINT := 0;
	iInit: LINT := 0;
	
	bElap: BOOL;
	tElap: TON;
	
	bStep: BOOL;
	tStep: TON;
	
	tHumidity_act: TON;
	bHumidity_act: BOOL;
	tHumidity_res: TON;
	bHumidity_res: BOOL;
	
	iMotor: INT;
	bMotor: BOOL;	
	tMotor: TON;
	
	iCounter: INT;
	
	bSound: BOOL;
END_VAR


IF EN = TRUE THEN

	IF Program_chamber[SL] = TRUE THEN
		
		CASE Program_chamber_status[SL] OF
			
			0:
				// Wainting init process
				
					Program_cycles[SL]:= 0;
					Program_steps[SL]:= 0;
					Program_elapsed[SL]:= 0;
					
					iInit:= 0;
					bElap:= 0;
					
					IF bSound = TRUE THEN
						bSound:= FALSE;
						Sound_activation[SL]:= FALSE;
					END_IF
					
			1: 
				// Init process	
				
					IF Program_elapsed[SL] = 0 THEN
						
						iEsti:= DT_TO_INT(TIME_TO_DT(Timer_convert(Program_estimated[SL], 'm'))) - DT_TO_LINT(DT#1970-01-01-00:00:00);
						iInit:= DT_TO_LINT(Program_process_init[SL]);
						Program_estimated_time[SL]:= LINT_TO_DT(iInit + iEsti);
					
						Program_chamber_status[SL]:= 2;
					END_IF
	
			2:
				//Chamber controller
				
					// Temperature core controller
						IF Core_temperature[SL] >= Recipe_core_temperature[SL] THEN
							Program_chamber_status[SL]:= 4;
						END_IF
				
					// Timer elapsed controller
						tElap(IN:= bElap, PT:= T#1M);
						
						IF bElap = FALSE THEN
							bElap:= TRUE;
						END_IF
						
						IF tElap.Q = TRUE THEN
							Program_elapsed[SL]:= Program_elapsed[SL] + 1;
							bElap:= FALSE;
						END_IF
						
					// Timer step controller
						tStep(IN:= bStep AND Program_steps[SL] < Recipe_steps[SL] AND Program_cycles[SL] < Recipe_cycles[SL], PT:= Timer_convert(Recipe_timer_step[SL, Program_steps[SL]],'m'));
						
						IF bStep = FALSE THEN
							bStep:= TRUE;
						END_IF
						
						IF Program_steps[SL] < Recipe_steps[SL] AND Program_cycles[SL] < Recipe_cycles[SL] THEN
							
							IF tStep.Q = TRUE THEN
								bStep:= FALSE;
								Program_steps[SL]:= Program_steps[SL] + 1;
							END_IF
	
						END_IF
						
						IF Program_steps[SL] = Recipe_steps[SL] AND Program_cycles[SL] < Recipe_cycles[SL] THEN
							Program_cycles[SL]:= Program_cycles[SL] + 1;
							IF Program_cycles[SL] < Recipe_cycles[SL] THEN
								Program_steps[SL]:= 0;
							END_IF
						END_IF
						
						IF Program_steps[SL] = Recipe_steps[SL] AND Program_cycles[SL] = Recipe_cycles[SL] THEN
							Program_chamber_status[SL]:= 5;
						END_IF
						
					// Temperature controller
					
						// Steam
							IF Temperature_control_system = FALSE THEN						
								IF 	Chamber_temperature[SL] < Recipe_chamber_temperature[SL, Program_steps[SL]] - Temperature_lower_hysteresis THEN
									Steam_valve_activation[SL]:= TRUE;
								END_IF
							
								IF 	Chamber_temperature[SL] > Recipe_chamber_temperature[SL, Program_steps[SL]] + Temperature_upper_hysteresis THEN
									Steam_valve_activation[SL]:= FALSE;
								END_IF
								
							END_IF
								
						// Burner
							IF Temperature_control_system = TRUE THEN
								
								IF 	Chamber_temperature[SL] < Recipe_chamber_temperature[SL, Program_steps[SL]] - Temperature_lower_hysteresis THEN
									Burner_activation[SL]:= TRUE;
								END_IF
							
								IF 	Chamber_temperature[SL] > Recipe_chamber_temperature[SL, Program_steps[SL]] + Temperature_upper_hysteresis THEN
									Burner_activation[SL]:= FALSE;
								END_IF
								
							END_IF
							
					// Humidity controller
						IF Temperature_control_system = FALSE THEN
							IF bHumidity_act = FALSE AND bHumidity_res = FALSE THEN
								IF Chamber_humidity[SL] < Recipe_chamber_humidity[SL, Program_steps[SL]] - Humidity_lower_hysteresis THEN
									bHumidity_act:= TRUE;
									Humidification_valve_activation[SL]:= TRUE;
								END_IF
							END_IF
							
							IF Chamber_humidity[SL] > Recipe_chamber_humidity[SL, Program_steps[SL]] + Humidity_upper_hysteresis THEN
								Humidification_valve_activation[SL]:= FALSE;
							END_IF
							
							IF tHumidity_act.Q = TRUE THEN
								bHumidity_act:= FALSE;
								bHumidity_res:= TRUE;
								Humidification_valve_activation[SL]:= FALSE;
							END_IF
							
							IF tHumidity_res.Q = TRUE THEN
								bHumidity_res:= FALSE;
							END_IF
							
							tHumidity_act(IN:= bHumidity_act, PT:= timer_convert(Timer_activation_humidification_valve, 's'));	
							tHumidity_res(IN:= bHumidity_res, PT:= timer_convert(timer_response_humidification_valve, 's'));
	
						END_IF
						
					// Chimney controller
						Chimney_activation[SL]:= Recipe_chamber_chimney[SL, Program_steps[SL]];
					
					// Smokehouse controller
						Smokehouse_activation[SL]:= Recipe_chamber_smokehouse[SL, Program_steps[SL]];
						
					// Motors controller
						tMotor(IN:= bMotor AND iMotor < Enabled_chamber_cars, PT:= Timer_convert(Timer_activation_motors, 's'));
						
						IF bMotor = FALSE THEN
							IF iMotor = 0 THEN
								Motor_activation[SL, iMotor]:= TRUE;
								iMotor:= iMotor + 1;
							END_IF
							bMotor:= TRUE;
						END_IF
						
						IF iMotor < Enabled_chamber_cars THEN
							
							IF tMotor.Q = TRUE THEN
								Motor_activation[SL, iMotor]:= TRUE;
								bMotor:= FALSE;
								iMotor:= iMotor + 1;
							END_IF
							
						END_IF
				
			3:
				// Proscess stalled
					iMotor:= 0;
					bMotor:= FALSE;
					
					FOR iCounter:= 0 TO Enabled_chamber_cars - 1 BY 1 DO
						Motor_activation[SL, iCounter]:= bMotor;
					END_FOR
				
			4:
				// Process terminated by the core temperature
					Steam_valve_activation[SL]:= FALSE;
					Humidification_valve_activation[SL]:= FALSE;
					Chimney_activation[SL]:= FALSE;
					Smokehouse_activation[SL]:= FALSE;

					iMotor:= 0;
					bMotor:= FALSE;
					
					FOR iCounter:= 0 TO Enabled_chamber_cars - 1 BY 1 DO
						Motor_activation[SL, iCounter]:= bMotor;
					END_FOR
			
					IF bSound = FALSE THEN
						Sound_activation[SL]:= TRUE;
						bSound:= TRUE;
					END_IF
					
			5:
				// Process terminated by the time
					Steam_valve_activation[SL]:= FALSE;
					Humidification_valve_activation[SL]:= FALSE;
					Chimney_activation[SL]:= FALSE;
					Smokehouse_activation[SL]:= FALSE;

					iMotor:= 0;
					bMotor:= FALSE;
					
					FOR iCounter:= 0 TO Enabled_chamber_cars - 1 BY 1 DO
						Motor_activation[SL, iCounter]:= bMotor;
					END_FOR
			
					IF bSound = FALSE THEN
						Sound_activation[SL]:= TRUE;
						bSound:= TRUE;
					END_IF
					
			6:
				// Process terminated by the user
					Steam_valve_activation[SL]:= FALSE;
					Humidification_valve_activation[SL]:= FALSE;
					Chimney_activation[SL]:= FALSE;
					Smokehouse_activation[SL]:= FALSE;

					iMotor:= 0;
					bMotor:= FALSE;
					
					FOR iCounter:= 0 TO Enabled_chamber_cars - 1 BY 1 DO
						Motor_activation[SL, iCounter]:= bMotor;
					END_FOR
				
			7:
				// Process terminated for failure
					Steam_valve_activation[SL]:= FALSE;
					Humidification_valve_activation[SL]:= FALSE;
					Chimney_activation[SL]:= FALSE;
					Smokehouse_activation[SL]:= FALSE;

					iMotor:= 0;
					bMotor:= FALSE;
					
					FOR iCounter:= 0 TO Enabled_chamber_cars - 1 BY 1 DO
						Motor_activation[SL, iCounter]:= bMotor;
					END_FOR
					
					IF bSound = FALSE THEN
						Sound_activation[SL]:= TRUE;
						bSound:= TRUE;
					END_IF
			
			8:
				// Chamber in failure
					Steam_valve_activation[SL]:= FALSE;
					Humidification_valve_activation[SL]:= FALSE;
					Chimney_activation[SL]:= FALSE;
					Smokehouse_activation[SL]:= FALSE;

					iMotor:= 0;
					bMotor:= FALSE;
					
					FOR iCounter:= 0 TO Enabled_chamber_cars - 1 BY 1 DO
						Motor_activation[SL, iCounter]:= bMotor;
					END_FOR
					
					IF bSound = FALSE THEN
						Sound_activation[SL]:= TRUE;
						bSound:= TRUE;
					END_IF
							
			9: 
				// Continuing the process
					Program_chamber_status[SL]:= 2;
					
					
		END_CASE
		
	END_IF

END_IF

END_FUNCTION_BLOCK

// Device/Application/Programs/Functions/Timer_convert
FUNCTION Timer_convert : TIME
VAR_INPUT
	Timer_int: INT;			//Set point OF timer
	Timer_uni: STRING;		//Timebase
END_VAR
VAR
	Timer_string: STRING;
END_VAR

	
Timer_string:= CONCAT('T#', INT_TO_STRING(Timer_int));
Timer_string:= CONCAT(Timer_string, Timer_uni);
Timer_convert:= STRING_TO_TIME(Timer_string);

END_FUNCTION

// Device/Application/Programs/Functions/Alarm_controller
FUNCTION_BLOCK Alarm_controller

VAR_INPUT
	EN: BOOL;	//Enable function
	SL: INT;	//Index of the chamber
END_VAR

VAR_OUTPUT
END_VAR

VAR
	tSteam_valte: TON;
	bSteam_valve: BOOL;
	rSteam_valve: REAL;
	
	tHumidity_valte: TON;
	bHumidity_valve: BOOL;
	iHumidity_valve: INT;
	
	tChimney_activation: TON;
	bChimney_activation: BOOL;
	bChimney_open: BOOL;
	bChimney_close: BOOL;
	
	iAlarm: INT;
END_VAR


//Burner_reset


IF EN = TRUE THEN
	
	// Analogs sensors
		// Core temperature sensor
			IF WORD_TO_REAL(Core_temperature_sensor[SL]) < 100.0 THEN
				Alarms_chambers_status[SL].00:= 1;
			ELSE
				Alarms_chambers_status[SL].00:= 0;
				IF WORD_TO_REAL(Core_temperature_sensor[SL]) > 1000.0 THEN
					Alarms_chambers_status[SL].01:= 1;
				ELSE
					IF WORD_TO_REAL(Core_temperature_sensor[SL]) >= 100.0 AND  WORD_TO_REAL(Core_temperature_sensor[SL]) <= 1000.0 THEN
						Alarms_chambers_status[SL].01:= 0;
					END_IF
				END_IF
			END_IF
		
		// Chamber temperature dry sensor
			IF WORD_TO_REAL(Chamber_temperature_dry_sensor[SL]) < 100.0 THEN
				Alarms_chambers_status[SL].02:= 1;
			ELSE
				Alarms_chambers_status[SL].02:= 0;
				IF WORD_TO_REAL(Chamber_temperature_dry_sensor[SL]) > 1000.0 THEN
					Alarms_chambers_status[SL].03:= 1;
				ELSE
					IF WORD_TO_REAL(Chamber_temperature_dry_sensor[SL]) >= 100.0 AND  WORD_TO_REAL(Chamber_temperature_dry_sensor[SL]) <= 1000.0 THEN
						Alarms_chambers_status[SL].03:= 0;
					END_IF
				END_IF
			END_IF
			
		// Chamber temperature wet sensor
			IF Temperature_control_system = FALSE THEN
				IF WORD_TO_REAL(Chamber_temperature_wet_sensor[SL]) < 100.0 THEN
					Alarms_chambers_status[SL].04:= 1;
				ELSE
					Alarms_chambers_status[SL].04:= 0;
					IF WORD_TO_REAL(Chamber_temperature_wet_sensor[SL]) < 100.0 THEN
						Alarms_chambers_status[SL].05:= 1;
					ELSE
						IF WORD_TO_REAL(Chamber_temperature_wet_sensor[SL]) >= 100.0 AND  WORD_TO_REAL(Chamber_temperature_wet_sensor[SL]) < 1000.0 THEN
							Alarms_chambers_status[SL].05:= 0;
						END_IF
					END_IF
				END_IF
			ELSE
				Alarms_chambers_status[SL].04:= 0;
				Alarms_chambers_status[SL].05:= 0;
			END_IF
			
	// Temperature control
		// Steam valve protection logic
			IF Temperature_control_system = FALSE THEN
				
				tSteam_valte(IN:= bSteam_valve, PT:= T#1M);
				
				IF Steam_valve_activation[SL] = TRUE AND bSteam_valve = FALSE THEN
					bSteam_valve:= TRUE;
					rSteam_valve:= Chamber_temperature[SL];
				END_IF
				
				IF tSteam_valte.Q = TRUE THEN
					bSteam_valve:= FALSE;
					
					IF rSteam_valve <= Chamber_temperature[SL] THEN
						Alarms_chambers_status[SL].06:= 1;
					ELSE
						Alarms_chambers_status[SL].06:= 0;
					END_IF
					
				END_IF
			
			ELSE
				Alarms_chambers_status[SL].06:= 0;
			END_IF
			
		// Burner protection circuit	
			IF Temperature_control_system = TRUE THEN
				Alarms_chambers_status[SL].07:= NOT Burner_protection[SL];
			END_IF
			
	// Humidity control
		// Humidification valve protection logic
			IF Temperature_control_system = FALSE THEN
				
				tHumidity_valte(IN:= bHumidity_valve, PT:= T#1M);
				
				IF Chamber_humidity[SL] < Recipe_chamber_humidity[SL, Program_steps[SL]] - Humidity_lower_hysteresis AND bHumidity_valve = FALSE THEN
					bHumidity_valve:= TRUE;
					iHumidity_valve:= Chamber_humidity[SL];
				END_IF
				
				IF tHumidity_valte.Q = TRUE THEN
					bHumidity_valve:= FALSE;
					
					IF iHumidity_valve <= Chamber_humidity[SL] THEN
						Alarms_chambers_status[SL].08:= 1;
					ELSE
						Alarms_chambers_status[SL].08:= 0;
					END_IF
					
				END_IF
				
			ELSE
				Alarms_chambers_status[SL].08:= 0;
			END_IF
		
	// Emergency chamber
		Alarms_chambers_status[SL].09:= NOT Emergency_chamber[SL];
		
	// Motor protection circuit
		Alarms_chambers_status[SL].10:= NOT Motor_protection[SL];
		
	// Temperature maximum
		IF Chamber_temperature[SL] >= Temperature_maximum THEN
			Alarms_chambers_status[SL].11:= 1;
		END_IF
		
		IF Chamber_temperature[SL] <= Temperature_maximum * 0.9 THEN
			Alarms_chambers_status[SL].11:= 0;
		END_IF
		
	// Chimney control
		tChimney_activation(IN:= bChimney_activation, PT:= T#5S);
		
		// Chimney open
			IF Chimney_activation[SL] = TRUE AND Higher_chimney_closed[SL] = TRUE AND Lower_chimney_closed[SL] = TRUE AND bChimney_open = FALSE THEN
				bChimney_open:= TRUE;
				bChimney_activation:= TRUE;
			END_IF
		
		// Chimney close
			IF Chimney_activation[SL] = FALSE AND Higher_chimney_open[SL] = TRUE AND Lower_chimney_open[SL] = TRUE AND bChimney_close = FALSE THEN
				bChimney_close:= TRUE;
				bChimney_activation:= TRUE;
			END_IF	
	
		IF tChimney_activation.Q = TRUE THEN
			bChimney_activation:= FALSE;
			
			IF bChimney_open = TRUE AND bChimney_close = FALSE THEN
				bChimney_open:= FALSE;
				
				IF Higher_chimney_closed[SL] = TRUE OR Lower_chimney_closed[SL] = TRUE OR Higher_chimney_open[SL] = FALSE OR Lower_chimney_open[SL] = FALSE THEN
					Alarms_chambers_status[SL].12:= 1;
				ELSE
					Alarms_chambers_status[SL].12:= 0;
				END_IF
				
			END_IF
			
			IF bChimney_close = TRUE AND bChimney_open = FALSE THEN
				bChimney_open:= FALSE;
				
				IF Higher_chimney_open[SL] = TRUE OR Lower_chimney_open[SL] = TRUE OR Higher_chimney_closed[SL] = FALSE OR Lower_chimney_closed[SL] = FALSE THEN
					Alarms_chambers_status[SL].13:= 1;
				ELSE
					Alarms_chambers_status[SL].13:= 0;
				END_IF
				
			END_IF
		END_IF
	
	// Smokehouse protection circuit
		Alarms_chambers_status[SL].14:= Smokehouse_protection[SL];
		
	// Alarm control
		IF Alarms_chambers_status[SL] > 0 AND Alarms_chambers_status[SL] <> iAlarm THEN
			
			IF Program_chamber_status[SL] > 0 AND Program_chamber_status[SL] < 8 THEN
				Program_chamber_status[SL]:= 7;
			ELSE
				Program_chamber_status[SL]:= 8;
			END_IF  
			
			Alarms_activation:= TRUE;
			iAlarm:= Alarms_chambers_status[SL];
		END_IF
		
		IF Alamrs_acknowledge = TRUE AND Alarms_activation = TRUE THEN
			Alamrs_acknowledge:= FALSE;
			Alarms_activation:= FALSE;
			Sound_activation[SL]:= FALSE;
			
			IF Alarms_chambers_status[SL] = 0 THEN
				Alarms_chambers_status[SL]:= 0;
				Program_chamber_status[SL]:= 0;
				iAlarm:= 0;
			END_IF
			
		END_IF
		
		IF Alarms_activation = TRUE THEN
			Sound_activation[SL]:= TRUE;
		END_IF
		
ELSE
	// Reset
		Alarms_chambers_status[SL]:= 0;
		
END_IF

END_FUNCTION_BLOCK

// Device/Application/Programs/Functions/Sound_controller
FUNCTION_BLOCK Sound_controller

VAR_INPUT
	EN: BOOL; 	//Enable function
END_VAR

VAR_OUTPUT
END_VAR

VAR
	iCounter: INT;
	
	bSound_Manual: BOOL;
	bSound_Process: BOOL;
	bSound_Alarm: BOOL;
	
	tSound_Process_On: TON;
	tSound_Process_Off: TON;
	tSound_Alarm_On: TON;
	tSound_Alarm_Off: TON;
	
END_VAR


IF EN = TRUE THEN
	
	bSound_Manual:= FALSE;
	bSound_Process:= FALSE;
	bSound_Alarm:= FALSE;
	
	FOR iCounter:= 0 TO Enabled_chambers - 1 BY 1 DO
		IF Program_chamber_status[iCounter] = 0 AND Sound_activation[iCounter] = TRUE THEN
			bSound_Manual:= TRUE;
		END_IF 
		
		IF Program_chamber_status[iCounter] > 3 AND Program_chamber_status[iCounter] < 6 AND Sound_activation[iCounter] = TRUE THEN
			bSound_Process:= TRUE;
		END_IF 
		
		IF Alarms_activation = TRUE AND Sound_activation[iCounter] = TRUE THEN
			bSound_Alarm:= TRUE;
		END_IF 
		
	END_FOR
	
	IF bSound_Alarm = TRUE THEN
		IF tSound_alarm_On.Q = TRUE AND tSound_Alarm_Off.Q = FALSE THEN
				Beeb_activation:= TRUE;
			ELSE
				Beeb_activation:= FALSE;
			END_IF
	ELSE
		IF bSound_Process = TRUE THEN
			IF tSound_Process_On.Q = TRUE AND tSound_Process_Off.Q = FALSE THEN
				Beeb_activation:= TRUE;
			ELSE
				Beeb_activation:= FALSE;
			END_IF
		ELSE
			IF bSound_Manual = TRUE THEN
				Beeb_activation:= TRUE;
			ELSE
				Beeb_activation:= FALSE;
			END_IF
		END_IF
	END_IF
	
	IF tSound_Alarm_Off.Q = TRUE THEN
		bSound_Alarm:= FALSE;
	END_IF
	
	IF tSound_Process_Off.Q = TRUE THEN
		bSound_Process:= FALSE;
	END_IF
	
	tSound_Alarm_On(IN:= bSound_Alarm, PT:= T#0.5S);
	tSound_Alarm_Off(IN:= tSound_Alarm_On.Q, PT:= T#0.5S);
	
	tSound_Process_On(IN:= bSound_Process, PT:= T#1S);	
	tSound_Process_Off(IN:= tSound_Process_On.Q, PT:= T#1S);
	
END_IF

END_FUNCTION_BLOCK
